{attribute 'GeneratedUsingTerminal: EL9188--0000'}
{attribute addProperty BoxType "EL9188--0000"}
{attribute addProperty Description "EL9188 Potential Connection, 16 x 24V"}
{attribute addProperty Physics "KK"}
{attribute addProperty Id "EL9188"}
{attribute addProperty CRC "2904417076"}
{attribute addProperty Size "0"}
TYPE EL9188_AD1DE334 EXTENDS EtcSlaveTerminalBase_947E5A46 :
STRUCT
END_STRUCT
END_TYPE

(* stored: Version 1.2.0.0, ProductVersion 3.1.4024.11
   DUT EL9188_AD1DE334: Id {027ee0aa-79db-477d-bd83-f997b759930b} *)
